// TwinCAT 3 PLC project Ex001
// ProgramVersion: 3.1.4024.0
// libraries:
//   Tc2_Standard, * (Beckhoff Automation GmbH)
//   Tc2_System, * (Beckhoff Automation GmbH)
//   Tc2_Utilities, * (Beckhoff Automation GmbH)
//   Tc3_Module, * (Beckhoff Automation GmbH)
// project tree:
//   DUTs/ E_EventType.TcDUT, ST_Event.TcDUT
//   / PlcTask.TcTTO
//   POUs/ EventLogger.TcPOU, FB_CsvPersistentEventStorage.TcPOU, FB_XmlPersistentEventStorage.TcPOU, F_UpdateEventTimestampWithSystemTime.TcPOU, I_PersistentEventStorage.TcIO, LightTower.TcIO, Log_Csv.TcPOU, MAIN.TcPOU, P_Warning.TcPOU
// real-time tasks:
//   TASK PlcTask: cycle T#10ms, priority 20, ADS port 350

CONFIGURATION Ex001
    RESOURCE PLC ON TwinCAT3
        TASK PlcTask(INTERVAL := T#10ms, PRIORITY := 20);
        PROGRAM MAIN WITH PlcTask : MAIN;
    END_RESOURCE
END_CONFIGURATION

// ---- DUTs/E_EventType.TcDUT
{attribute 'qualified_only'}
{attribute 'strict'}
{attribute 'to_string'}
TYPE E_EventType :
(
	Alarm := 0,
	Message := 1
);
END_TYPE

// ---- DUTs/ST_Event.TcDUT
TYPE ST_Event :
STRUCT
	eEventType : E_EventType;
	eEventSeverity : TcEventSeverity;
	nEventIdentity : UDINT;
	sEventText : STRING(255);
	dtTimestamp : DATE_AND_TIME;
END_STRUCT
END_TYPE

// ---- POUs/I_PersistentEventStorage.TcIO
INTERFACE I_PersistentEventStorage

METHOD StoreEvent
VAR_INPUT
	stEvent : ST_Event;
END_VAR
END_METHOD

END_INTERFACE

// ---- POUs/LightTower.TcIO
INTERFACE LightTower

METHOD Blink : BOOL
VAR_INPUT
	On : BOOL;
END_VAR
END_METHOD

METHOD OnOff
VAR_INPUT
	On : BOOL;
END_VAR
END_METHOD

END_INTERFACE

// ---- POUs/MAIN.TcPOU
PROGRAM MAIN
VAR
	//st_Fupdate : ST_Event;
	btOne : BOOL := FALSE;
	
	// Trang thai cho su kien
	eEventType : E_EventType := E_EventType.Alarm;
	eEventSeverity : TcEventSeverity := TcEventSeverity.Error;
	nEventIdentity : UDINT := 32;
	sEventText : STRING(255) := 'Status';
	
	XmlPersistentEventStorage : FB_XmlPersistentEventStorage;
	EventLogger : EventLogger(XmlPersistentEventStorage);
	
END_VAR

// P_Warning();
(*
IF NOT btOne THEN
	F_UpdateEventTimestampWithSystemTime(stEvent := st_Fupdate);
	btOne := TRUE;
END_IF
*)

(*IF btOne THEN
	EventLogger.AddEvent(eEventType, eEventSeverity, nEventIdentity, sEventText);
	btOne := FALSE;
END_IF*)
Log_Csv();

END_PROGRAM

// ---- POUs/FB_XmlPersistentEventStorage.TcPOU
FUNCTION_BLOCK FB_XmlPersistentEventStorage IMPLEMENTS I_PersistentEventStorage
VAR_INPUT
END_VAR
VAR_OUTPUT
END_VAR
VAR
END_VAR

//

METHOD StoreEvent
VAR_INPUT
	stEvent	: ST_Event;
END_VAR
END_METHOD

END_FUNCTION_BLOCK

// ---- POUs/EventLogger.TcPOU
FUNCTION_BLOCK EventLogger
VAR
	EventBuffer : ARRAY[1..Maxinum_size_event_buffer] OF ST_Event;
	CurrentEventBufferIndex : INT := 0;
	
	_PersistentEventStorage : I_PersistentEventStorage;
END_VAR
VAR CONSTANT
	Maxinum_size_event_buffer : INT := 100;
END_VAR

(* Returns TRUE if add was succesful and FALSE if buffer is full *)
METHOD PUBLIC AddEvent : BOOL
VAR_INPUT
	eEventType : E_EventType;
	eEventSeverity : TcEventSeverity;
	nEventIdentity : UDINT;
	sEventText : STRING(255);
END_VAR
IF NOT IsEventBufferFull() THEN
	CurrentEventBufferIndex := CurrentEventBufferIndex + 1;
	EventBuffer[CurrentEventBufferIndex].eEventType := eEventType;
	EventBuffer[CurrentEventBufferIndex].eEventSeverity := eEventSeverity;
	EventBuffer[CurrentEventBufferIndex].nEventIdentity := nEventIdentity;
	EventBuffer[CurrentEventBufferIndex].sEventText := sEventText;
	F_UpdateEventTimestampWithSystemTime(stEvent := EventBuffer[CurrentEventBufferIndex]);
	AddEvent := TRUE;
ELSE
	AddEvent := FALSE;		
END_IF


// Event Persistently

_PersistentEventStorage.StoreEvent(stEvent := EventBuffer[CurrentEventBufferIndex]);
END_METHOD

METHOD FB_init : BOOL
VAR_INPUT
	bInitRetains : BOOL; // if TRUE, the retain variables are initialized (warm start / cold start)
	bInCopyCode : BOOL;  // if TRUE, the instance afterwards gets moved into the copy code (online change)
	
	iPersistentEventStorage : I_PersistentEventStorage;
END_VAR
_PersistentEventStorage := iPersistentEventStorage;
END_METHOD

METHOD PRIVATE IsEventBufferFull : BOOL
IF (CurrentEventBufferIndex + 1) > Maxinum_size_event_buffer THEN 
	IsEventBufferFull := TRUE;
ELSE 
	IsEventBufferFull := FALSE;
END_IF
END_METHOD

END_FUNCTION_BLOCK

// ---- POUs/F_UpdateEventTimestampWithSystemTime.TcPOU
FUNCTION F_UpdateEventTimestampWithSystemTime
VAR_INPUT
	stEvent : Reference to ST_Event;
END_VAR
VAR
	fbGETSYSTEMTIME : GETSYSTEMTIME;
	
	stFileTime : T_FILETIME;
END_VAR

fbGETSYSTEMTIME(timeLoDW => stFileTime.dwLowDateTime,
				timeHiDW => stFileTIme.dwHighDateTime);
stEvent.dtTimestamp := FILETIME_TO_DT(fileTime := stFileTime);

END_FUNCTION

// ---- POUs/Log_Csv.TcPOU
PROGRAM Log_Csv
VAR
	trig1 : BOOL := FALSE;
	// Trang thai cho su kien
	eEventType : E_EventType := E_EventType.Alarm;
	eEventSeverity : TcEventSeverity := TcEventSeverity.Error;
	nEventIdentity : UDINT := 32;
	sEventText : STRING(255) := 'Status';
	nEventID : UDINT;
	
	CsvPersistentEventStorage : FB_CsvPersistentEventStorage;
	EventLogger : EventLogger(CsvPersistentEventStorage);
END_VAR


IF trig1 THEN
    // Gọi method GetEventTextByID từ CsvPersistentEventStorage để lấy text dựa trên nEventID
    sEventText := CsvPersistentEventStorage.GetEventTextByID(nEventID);
    // Ghi log sự kiện với thông tin đã cập nhật
    EventLogger.AddEvent(eEventType, eEventSeverity, nEventIdentity, sEventText);
    trig1 := FALSE;
END_IF;
CsvPersistentEventStorage();

END_PROGRAM

// ---- POUs/FB_CsvPersistentEventStorage.TcPOU
FUNCTION_BLOCK FB_CsvPersistentEventStorage IMPLEMENTS I_PersistentEventStorage
VAR
	fbFileOpen : FB_FileOpen := (sPathName :='D:\folderData\Twincat\TestCSV\Event20.log', nMode := FOPEN_MODEAPPEND OR FOPEN_MODETEXT);
	fbFilePuts : FB_FilePuts;
	fbFileClose : FB_FileClose;
	eWriteState : (FILE_OPEN_TRIGGER,FILE_OPEN, WAIT_FOR_EVENT, WRITE_EVENT_TRIGGER, WRITE_EVENT, FILE_CLOSE_TRIGGER, FILE_CLOSE, ERROR);
	stEventWrittenToFile : ST_Event;
	
	CsvString : T_MaxString;
END_VAR

(*
	S1: FILE_OPEN_TRIGGER: Kích hoạt mở file.
	S2: FILE_OPEN: Kiểm tra trạng thái mở file, xử lý lỗi nếu có.
	S3: WAIT_FOR_EVENT: Chờ sự kiện cần ghi.
	S4: WRITE_EVENT_TRIGGER: Tạo chuỗi CSV và kích hoạt ghi.
	S5: WRITE_EVENT: Ghi dữ liệu vào file, kiểm tra lỗi khi ghi.
	S6: FILE_CLOSE_TRIGGER: Kích hoạt đóng file.
	S7: FILE_CLOSE: Đóng file và quay lại trạng thái mở file.
	S8: ERROR: Xử lý lỗi, không thực hiện hành động khác.
*)

CASE eWriteState OF
    // Lua chon hanh dong dua vao trang thai hien tai cua eWriteState
    
    FILE_OPEN_TRIGGER :
        fbFileOpen(bExecute := TRUE);
        // Bat dau mo file bang cach kich hoat fbFileOpen
        eWriteState := FILE_OPEN;
        // Chuyen sang trang thai FILE_OPEN de xu ly tiep

    FILE_OPEN :
        fbFileOpen(bExecute := FALSE);
        // Ngung kich hoat fbFileOpen sau khi da goi lenh mo file
        IF fbFileOpen.bError THEN
            eWriteState := ERROR;
            // Neu co loi xay ra trong qua trinh mo file, chuyen sang trang thai ERROR
        ELSIF NOT fbFileOpen.bBusy AND fbFileOpen.hFile <> 0 THEN
            eWriteState := WAIT_FOR_EVENT;
            // Neu file mo thanh cong va khong con ban, chuyen sang trang thai WAIT_FOR_EVENT
        END_IF

    WAIT_FOR_EVENT:
        // Do no thing

    WRITE_EVENT_TRIGGER :
        CsvString := CreateCsvString(stEvent := stEventWrittenToFile);
        // Tao chuoi CSV dua tren du lieu su kien stEventWrittenToFile
        fbFilePuts(bExecute := TRUE,
                   sLine := CsvString,
                   hFile := fbFileOpen.hFile);
        // Kich hoat fbFilePuts de ghi chuoi CSV vao file
        eWriteState := WRITE_EVENT;
        // Chuyen sang trang thai WRITE_EVENT de xu ly ghi du lieu

    WRITE_EVENT :
        fbFilePuts(bExecute := FALSE);
        // Ngung kich hoat fbFilePuts sau khi goi lenh ghi du lieu
        IF fbFilePuts.bError THEN
            eWriteState := ERROR;
            // Neu co loi trong qua trinh ghi, chuyen sang trang thai ERROR
        ELSIF NOT fbFilePuts.bBusy THEN
            eWriteState := FILE_CLOSE_TRIGGER;
            // Neu ghi thanh cong va hoan tat, chuyen sang trang thai FILE_CLOSE_TRIGGER
        END_IF

    FILE_CLOSE_TRIGGER :
        fbFileClose(bExecute := TRUE,
                    hFile := fbFileOpen.hFile);
        // Kich hoat fbFileClose de dong file
        eWriteState := FILE_CLOSE;
        // Chuyen sang trang thai FILE_CLOSE de xu ly tiep

    FILE_CLOSE :
        fbFileClose(bExecute := FALSE);
        // Ngung kich hoat fbFileClose sau khi goi lenh dong file
        IF fbFileClose.bError THEN
            eWriteState := ERROR;
            // Neu co loi trong qua trinh dong file, chuyen sang trang thai ERROR
        ELSIF NOT fbFileClose.bBusy THEN
            eWriteState := FILE_OPEN_TRIGGER;
            // Neu dong file thanh cong, quay lai trang thai FILE_OPEN_TRIGGER
        END_IF

    ERROR:
        // Do no thing

END_CASE

METHOD PRIVATE CreateCsvString : T_MaxString
VAR_INPUT
	stEvent : REFERENCE TO ST_Event;
END_VAR
VAR
	TempString : T_MaxString;
END_VAR
TempString := TO_STRING(stEvent.eEventType);
TempString := CONCAT(STR1 := TempString, STR2 := ',');
TempString := CONCAT(STR1 := TempString, STR2 := TO_STRING(stEvent.eEventSeverity));
TempString := CONCAT(STR1 := TempString, STR2 := ',');
TempString := CONCAT(STR1 := TempString, STR2 := TO_STRING(stEvent.nEventIdentity));
TempString := CONCAT(STR1 := TempString, STR2 := ',');
TempString := CONCAT(STR1 := TempString, STR2 := stEvent.sEventText);
TempString := CONCAT(STR1 := TempString, STR2 := ',');
TempString := CONCAT(STR1 := TempString, STR2 := TO_STRING(stEvent.dtTimestamp));
TempString := CONCAT(STR1 := TempString, STR2 := '$n');

CreateCsvString := TempString;
END_METHOD

METHOD PUBLIC GetEventTextByID : T_MaxString
VAR_INPUT
	nID : UDINT; 
END_VAR
VAR
	sResult : T_MaxString; 
END_VAR
CASE nID OF
    1: sResult := 'Error: Sensor not connected';
    2: sResult := 'Warning: Temperature high';
    3: sResult := 'Info: System started';
	4: sResult := 'Hello everyone';
    ELSE
        sResult := 'Unknown Event';
END_CASE;

GetEventTextByID := sResult;
END_METHOD

METHOD StoreEvent
VAR_INPUT
	stEvent	: ST_Event;
END_VAR
// T132S
IF eWriteState = WAIT_FOR_EVENT THEN
	eWriteState := WRITE_EVENT_TRIGGER;
	stEventWrittenToFile := stEvent;
END_IF
END_METHOD

END_FUNCTION_BLOCK

// ---- POUs/P_Warning.TcPOU
PROGRAM P_Warning
VAR
	btRun : BOOL := FALSE;
END_VAR

IF NOT btRun THEN
	ADSLOGSTR(msgCtrlMask := ADSLOG_MSGTYPE_ERROR OR ADSLOG_MSGTYPE_LOG,
			  msgFmtStr := 'hi Thinh',
			  strArg := '');
	btRun := TRUE;
END_IF

END_PROGRAM
